(* Schneider Machine Expert - Basic project es3_4pompe_3max_6soglie_spegnimento_graduale_semplice, file version 3.0.0.0 *)
(* ProjectInformations: Name=New project *)

HARDWARE
  Cpu 0: TM221C40R
  EthernetConfiguration: NetworkName=M221, IpAllocationMode=FixedAddress, IpAddress=0.0.0.0, SubnetMask=0.0.0.0
  SerialLineConfiguration: Baud=Baud19200, Parity=ParityEven, DataBits=DataBits8, StopBits=StopBits1, PhysicalMedium=PhysicalMediumRs485, TransmissionMode=TransmissionModeModbusRtu, SlaveId=1, Addressing=SlaveAddressing
  MastTask: UsePeriodScanMode=false, PeriodScan=100
  FastTask: Period=255
  CpuBehavior: StartingMode=StartAsPreviousState, AutoSaveRamOnEeprom=true, WatchdogPeriod=250

SYMBOLS  (address, symbol, comment, settings)
  %M0       P1_USABILE
  %M1       P2_USABILE
  %M2       P1_COMANDATA  "Stesso valore di P1_CMD. Permette di identificare gli edges, visto che P1_CMD non può farlo."
  %M3       P2_COMANDATA  "Stesso valore di P2_CMD. Permette di identificare gli edges, visto che P2_CMD non può farlo."
  %M4       P3_USABILE
  %M5       P4_USABILE
  %M6       P3_COMANDATA
  %M7       P4_COMANDATA
  %M8       ESISTE_PROX_POMPA_CON_MINOR_ORE  "Nel loop, può non esistere una prossima pompa usabile e non comandata con il minor numero ore."
  %M9       ORA_E_00  "E' mezzanotte?"
  %M10      DECISO_ORDINE  "In intervallo in cui alternare le pompe per altern. giorn., è stata deciso quale sarà prossima pompa con minor ore?"
  %M11      PRIMA_POMPA_COMANDATA  "La prima pompa dell'ordine è stata effettivamente comandata quando serviva?"
  %M12      SECONDA_POMPA_COMANDATA  "La seconda pompa dell'ordine è stata effettivamente comandata quando serviva?"
  %M13      TERZA_POMPA_COMANDATA  "La terza pompa dell'ordine è stata effettivamente comandata quando serviva?"
  %S6       SB_TB1S  "Time base of 1 s generated by an internal clock"
  %MW0      NUM_POMPE_DA_COMANDARE  "Numero di pompe da comandare in base alle soglie raggiunte."
  %MW1      NUM_POMPE_COMANDATE  "Numero di pompe effettivamente comandate, in base alle loro disponibilità."
  %MW2      NUM_POMPE  "Numero di pompe totali."
  %MW3      ULTIMO_MINOR_SECONDI_LAVORATI  "Ultimi secondi lavorati più piccoli (valore temporaneo, da usare solo nel loop)."
  %MW4      PROSSIMA_POMPA_DA_COMANDARE  "Numero da 1 a NUM_POMPE che indica la prossima pompa da comandare."
  %MW5      POMPA_ATTUALE_LOOP  "Pompa attuale nel loop."
  %MW6      NUM_POMPE_COMANDATE_MAX  "Num"
  %MW7      CONTA_POMPE_COMANDATE_MAX  "Da usare in loop e da resettare.  Assume il valore da 1 fino a NUM_POMPE_COMANDATE_MAX."
  %MW8      ORDINE_PRIMA_POMPA
  %MW9      ORDINE_SECONDA_POMPA
  %MW10     ORDINE_TERZA_POMPA
  %C0       CONTATORE_P1_SECONDI_LAVORATI  [Preset=0]
  %C1       CONTATORE_P2_SECONDI_LAVORATI  [Preset=0]
  %C2       CONTATORE_P3_SECONDI_LAVORATI  [Preset=0]
  %C3       CONTATORE_P4_SECONDI_LAVORATI  [Preset=0]
  %I0.0     P1_AUTO
  %I0.1     P1_MOTO
  %I0.2     P1_ANOMALIA
  %I0.3     P2_AUTO
  %I0.4     P2_MOTO
  %I0.5     P2_ANOMALIA
  %I0.6     LVL_MIN1
  %I0.7     LVL_MAX1
  %I0.8     LVL_MAX2
  %I0.9     P3_AUTO
  %I0.10    P3_MOTO
  %I0.11    P3_ANOMALIA
  %I0.12    P4_AUTO
  %I0.13    P4_MOTO
  %I0.14    P4_ANOMALIA
  %I0.15    LVL_MAX3
  %I0.16    LVL_MIN2
  %I0.17    LVL_MIN3
  %Q0.0     P1_CMD
  %Q0.1     P2_CMD
  %Q0.2     P3_CMD
  %Q0.3     P4_CMD

POU Main
  (* SectionNumber=1 *)

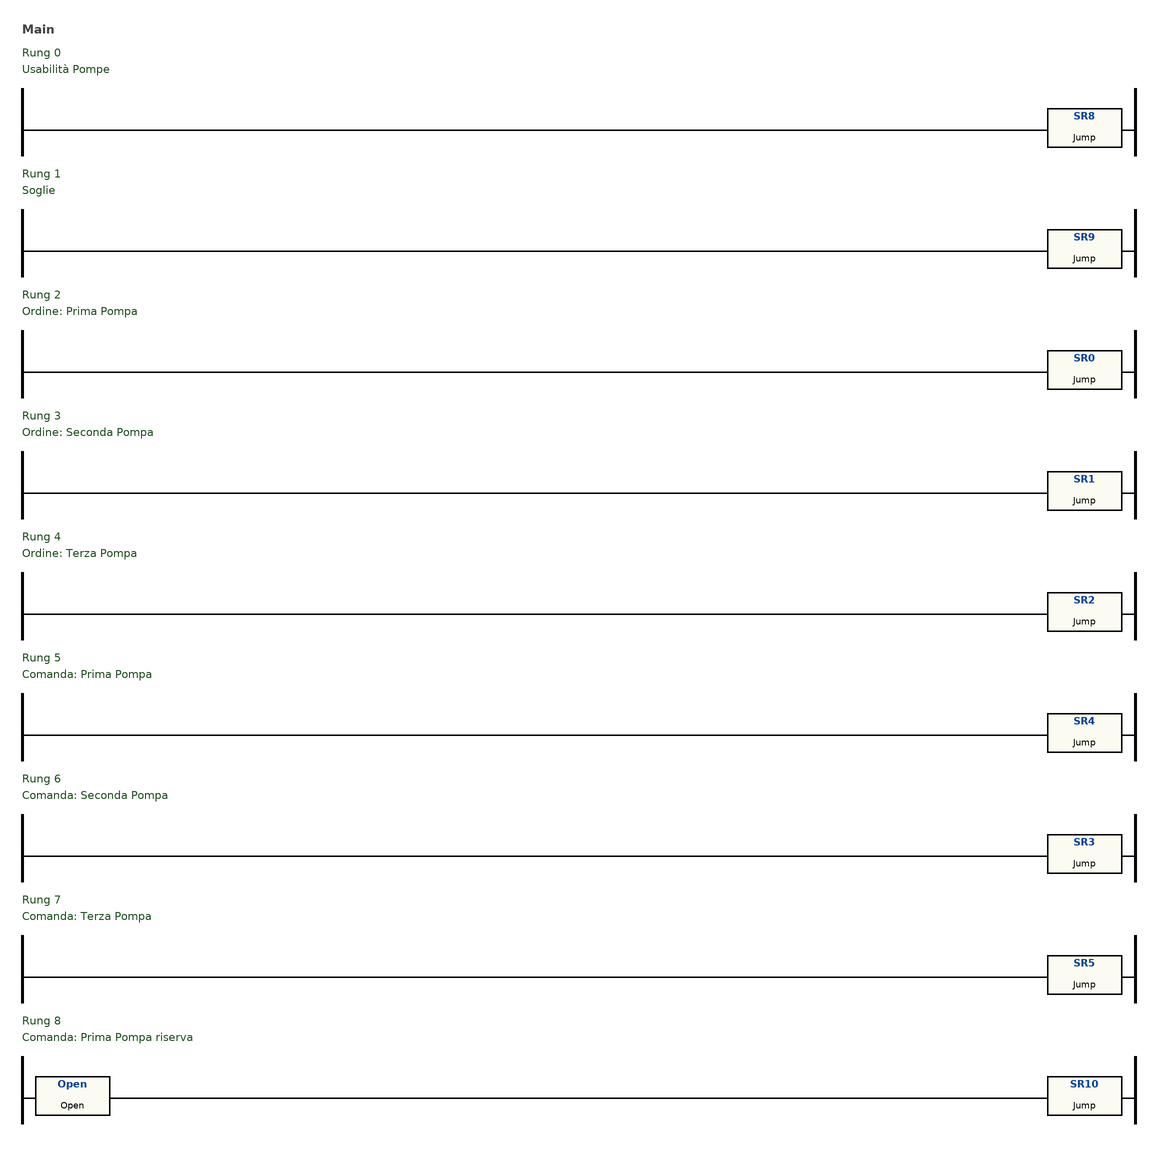

// Rung 0
// Usabilità Pompe
  LD 1
  SR8
  // as ST:
  //   SR8();

// Rung 1
// Soglie
  LD 1
  SR9
  // as ST:
  //   SR9();

// Rung 2
// Ordine: Prima Pompa
  LD 1
  SR0
  // as ST:
  //   SR0();

// Rung 3
// Ordine: Seconda Pompa
  LD 1
  SR1
  // as ST:
  //   SR1();

// Rung 4
// Ordine: Terza Pompa
  LD 1
  SR2
  // as ST:
  //   SR2();

// Rung 5
// Comanda: Prima Pompa
  LD 1
  SR4
  // as ST:
  //   SR4();

// Rung 6
// Comanda: Seconda Pompa
  LD 1
  SR3
  // as ST:
  //   SR3();

// Rung 7
// Comanda: Terza Pompa
  LD 1
  SR5
  // as ST:
  //   SR5();

// Rung 8
// Comanda: Prima Pompa riserva
  LD 0
  SR10
  // as ST:
  //   IF FALSE THEN SR10(); END_IF;

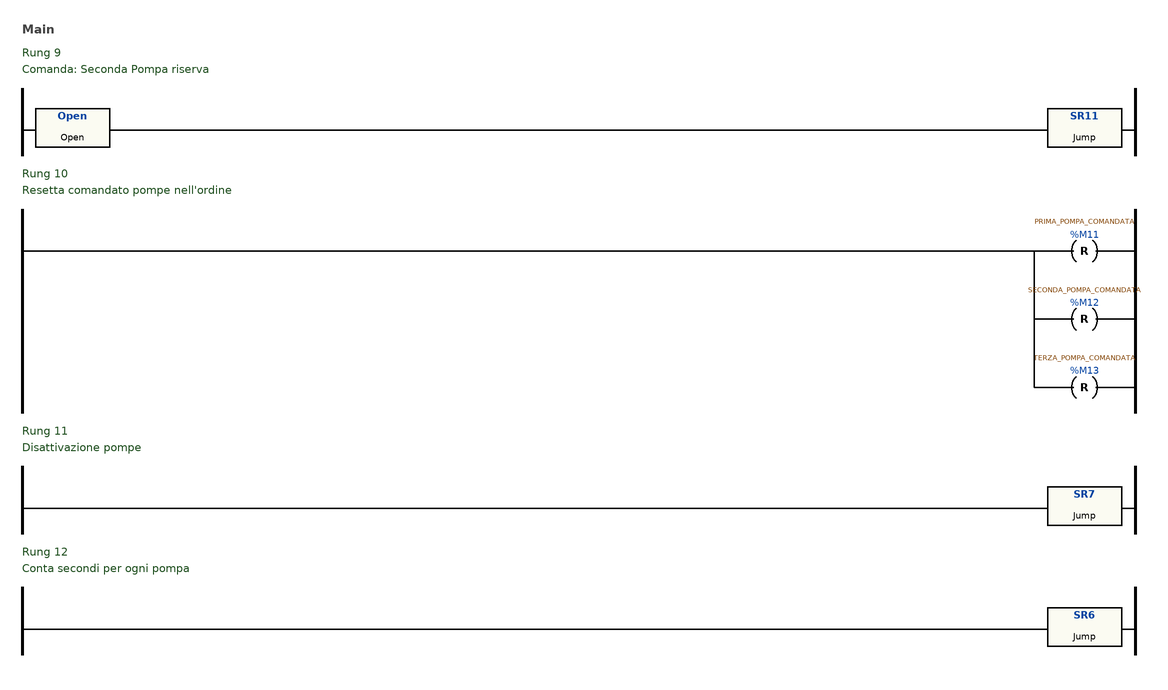

// Rung 9
// Comanda: Seconda Pompa riserva
  LD 0
  SR11
  // as ST:
  //   IF FALSE THEN SR11(); END_IF;

// Rung 10
// Resetta comandato pompe nell'ordine
  LD 1
  R %M11                  (* PRIMA_POMPA_COMANDATA *)
  R %M12                  (* SECONDA_POMPA_COMANDATA *)
  R %M13                  (* TERZA_POMPA_COMANDATA *)
  // as ST:
  //   PRIMA_POMPA_COMANDATA := FALSE;
  //   SECONDA_POMPA_COMANDATA := FALSE;
  //   TERZA_POMPA_COMANDATA := FALSE;

// Rung 11
// Disattivazione pompe
  LD 1
  SR7
  // as ST:
  //   SR7();

// Rung 12
// Conta secondi per ogni pompa
  LD 1
  SR6
  // as ST:
  //   SR6();

Subroutine Ordine: Prima Pompa
  (* SectionNumber=2, Number=0 *)

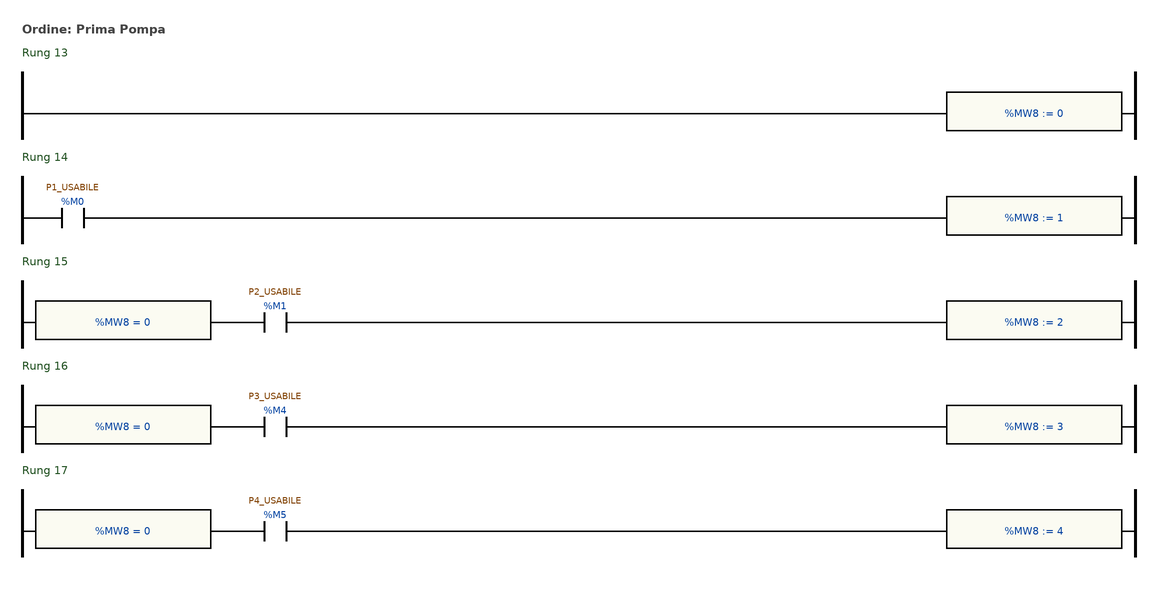

// Rung 13
  LD 1
  [ %MW8 := 0 ]           (* ORDINE_PRIMA_POMPA *)
  // as ST:
  //   ORDINE_PRIMA_POMPA := 0;

// Rung 14
  LD %M0                  (* P1_USABILE *)
  [ %MW8 := 1 ]           (* ORDINE_PRIMA_POMPA *)
  // as ST:
  //   IF P1_USABILE THEN ORDINE_PRIMA_POMPA := 1; END_IF;

// Rung 15
  LD [ %MW8 = 0 ]         (* ORDINE_PRIMA_POMPA *)
  AND %M1                 (* P2_USABILE *)
  [ %MW8 := 2 ]           (* ORDINE_PRIMA_POMPA *)
  // as ST:
  //   IF ORDINE_PRIMA_POMPA = 0 AND P2_USABILE THEN ORDINE_PRIMA_POMPA := 2; END_IF;

// Rung 16
  LD [ %MW8 = 0 ]         (* ORDINE_PRIMA_POMPA *)
  AND %M4                 (* P3_USABILE *)
  [ %MW8 := 3 ]           (* ORDINE_PRIMA_POMPA *)
  // as ST:
  //   IF ORDINE_PRIMA_POMPA = 0 AND P3_USABILE THEN ORDINE_PRIMA_POMPA := 3; END_IF;

// Rung 17
  LD [ %MW8 = 0 ]         (* ORDINE_PRIMA_POMPA *)
  AND %M5                 (* P4_USABILE *)
  [ %MW8 := 4 ]           (* ORDINE_PRIMA_POMPA *)
  // as ST:
  //   IF ORDINE_PRIMA_POMPA = 0 AND P4_USABILE THEN ORDINE_PRIMA_POMPA := 4; END_IF;

Subroutine Ordine: Seconda Pompa
  (* SectionNumber=3, Number=1 *)

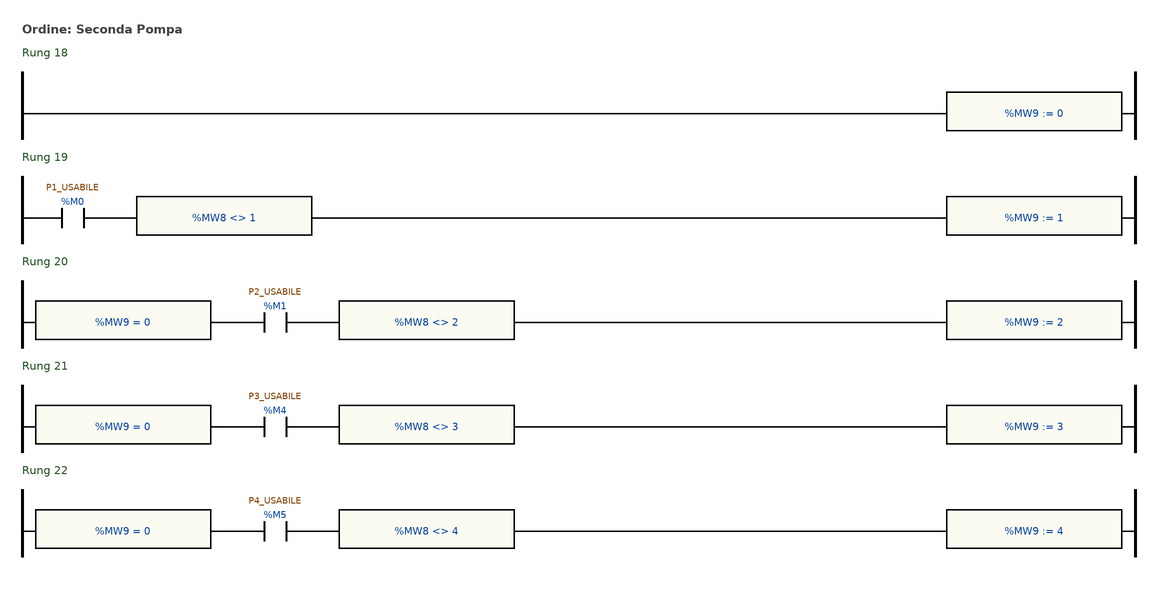

// Rung 18
  LD 1
  [ %MW9 := 0 ]           (* ORDINE_SECONDA_POMPA *)
  // as ST:
  //   ORDINE_SECONDA_POMPA := 0;

// Rung 19
  LD %M0                  (* P1_USABILE *)
  AND [ %MW8 <> 1 ]       (* ORDINE_PRIMA_POMPA *)
  [ %MW9 := 1 ]           (* ORDINE_SECONDA_POMPA *)
  // as ST:
  //   IF P1_USABILE AND ORDINE_PRIMA_POMPA <> 1 THEN ORDINE_SECONDA_POMPA := 1; END_IF;

// Rung 20
  LD [ %MW9 = 0 ]         (* ORDINE_SECONDA_POMPA *)
  AND %M1                 (* P2_USABILE *)
  AND [ %MW8 <> 2 ]       (* ORDINE_PRIMA_POMPA *)
  [ %MW9 := 2 ]           (* ORDINE_SECONDA_POMPA *)
  // as ST:
  //   IF ORDINE_SECONDA_POMPA = 0 AND P2_USABILE AND ORDINE_PRIMA_POMPA <> 2 THEN ORDINE_SECONDA_POMPA := 2; END_IF;

// Rung 21
  LD [ %MW9 = 0 ]         (* ORDINE_SECONDA_POMPA *)
  AND %M4                 (* P3_USABILE *)
  AND [ %MW8 <> 3 ]       (* ORDINE_PRIMA_POMPA *)
  [ %MW9 := 3 ]           (* ORDINE_SECONDA_POMPA *)
  // as ST:
  //   IF ORDINE_SECONDA_POMPA = 0 AND P3_USABILE AND ORDINE_PRIMA_POMPA <> 3 THEN ORDINE_SECONDA_POMPA := 3; END_IF;

// Rung 22
  LD [ %MW9 = 0 ]         (* ORDINE_SECONDA_POMPA *)
  AND %M5                 (* P4_USABILE *)
  AND [ %MW8 <> 4 ]       (* ORDINE_PRIMA_POMPA *)
  [ %MW9 := 4 ]           (* ORDINE_SECONDA_POMPA *)
  // as ST:
  //   IF ORDINE_SECONDA_POMPA = 0 AND P4_USABILE AND ORDINE_PRIMA_POMPA <> 4 THEN ORDINE_SECONDA_POMPA := 4; END_IF;

Subroutine Ordine: Terza Pompa
  (* SectionNumber=4, Number=2 *)

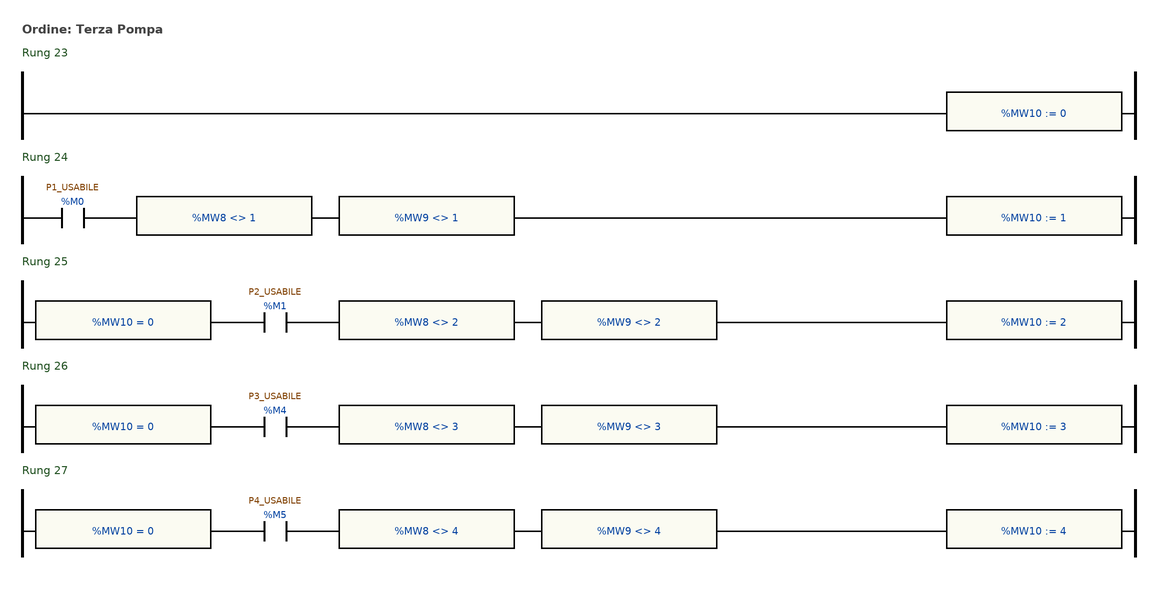

// Rung 23
  LD 1
  [ %MW10 := 0 ]          (* ORDINE_TERZA_POMPA *)
  // as ST:
  //   ORDINE_TERZA_POMPA := 0;

// Rung 24
  LD %M0                  (* P1_USABILE *)
  AND [ %MW8 <> 1 ]       (* ORDINE_PRIMA_POMPA *)
  AND [ %MW9 <> 1 ]       (* ORDINE_SECONDA_POMPA *)
  [ %MW10 := 1 ]          (* ORDINE_TERZA_POMPA *)
  // as ST:
  //   IF P1_USABILE AND ORDINE_PRIMA_POMPA <> 1 AND ORDINE_SECONDA_POMPA <> 1 THEN ORDINE_TERZA_POMPA := 1; END_IF;

// Rung 25
  LD [ %MW10 = 0 ]        (* ORDINE_TERZA_POMPA *)
  AND %M1                 (* P2_USABILE *)
  AND [ %MW8 <> 2 ]       (* ORDINE_PRIMA_POMPA *)
  AND [ %MW9 <> 2 ]       (* ORDINE_SECONDA_POMPA *)
  [ %MW10 := 2 ]          (* ORDINE_TERZA_POMPA *)
  // as ST:
  //   IF ORDINE_TERZA_POMPA = 0 AND P2_USABILE AND ORDINE_PRIMA_POMPA <> 2 AND ORDINE_SECONDA_POMPA <> 2 THEN ORDINE_TERZA_POMPA := 2; END_IF;

// Rung 26
  LD [ %MW10 = 0 ]        (* ORDINE_TERZA_POMPA *)
  AND %M4                 (* P3_USABILE *)
  AND [ %MW8 <> 3 ]       (* ORDINE_PRIMA_POMPA *)
  AND [ %MW9 <> 3 ]       (* ORDINE_SECONDA_POMPA *)
  [ %MW10 := 3 ]          (* ORDINE_TERZA_POMPA *)
  // as ST:
  //   IF ORDINE_TERZA_POMPA = 0 AND P3_USABILE AND ORDINE_PRIMA_POMPA <> 3 AND ORDINE_SECONDA_POMPA <> 3 THEN ORDINE_TERZA_POMPA := 3; END_IF;

// Rung 27
  LD [ %MW10 = 0 ]        (* ORDINE_TERZA_POMPA *)
  AND %M5                 (* P4_USABILE *)
  AND [ %MW8 <> 4 ]       (* ORDINE_PRIMA_POMPA *)
  AND [ %MW9 <> 4 ]       (* ORDINE_SECONDA_POMPA *)
  [ %MW10 := 4 ]          (* ORDINE_TERZA_POMPA *)
  // as ST:
  //   IF ORDINE_TERZA_POMPA = 0 AND P4_USABILE AND ORDINE_PRIMA_POMPA <> 4 AND ORDINE_SECONDA_POMPA <> 4 THEN ORDINE_TERZA_POMPA := 4; END_IF;

Subroutine Comanda: Prima Pompa
  (* SectionNumber=5, Number=4 *)

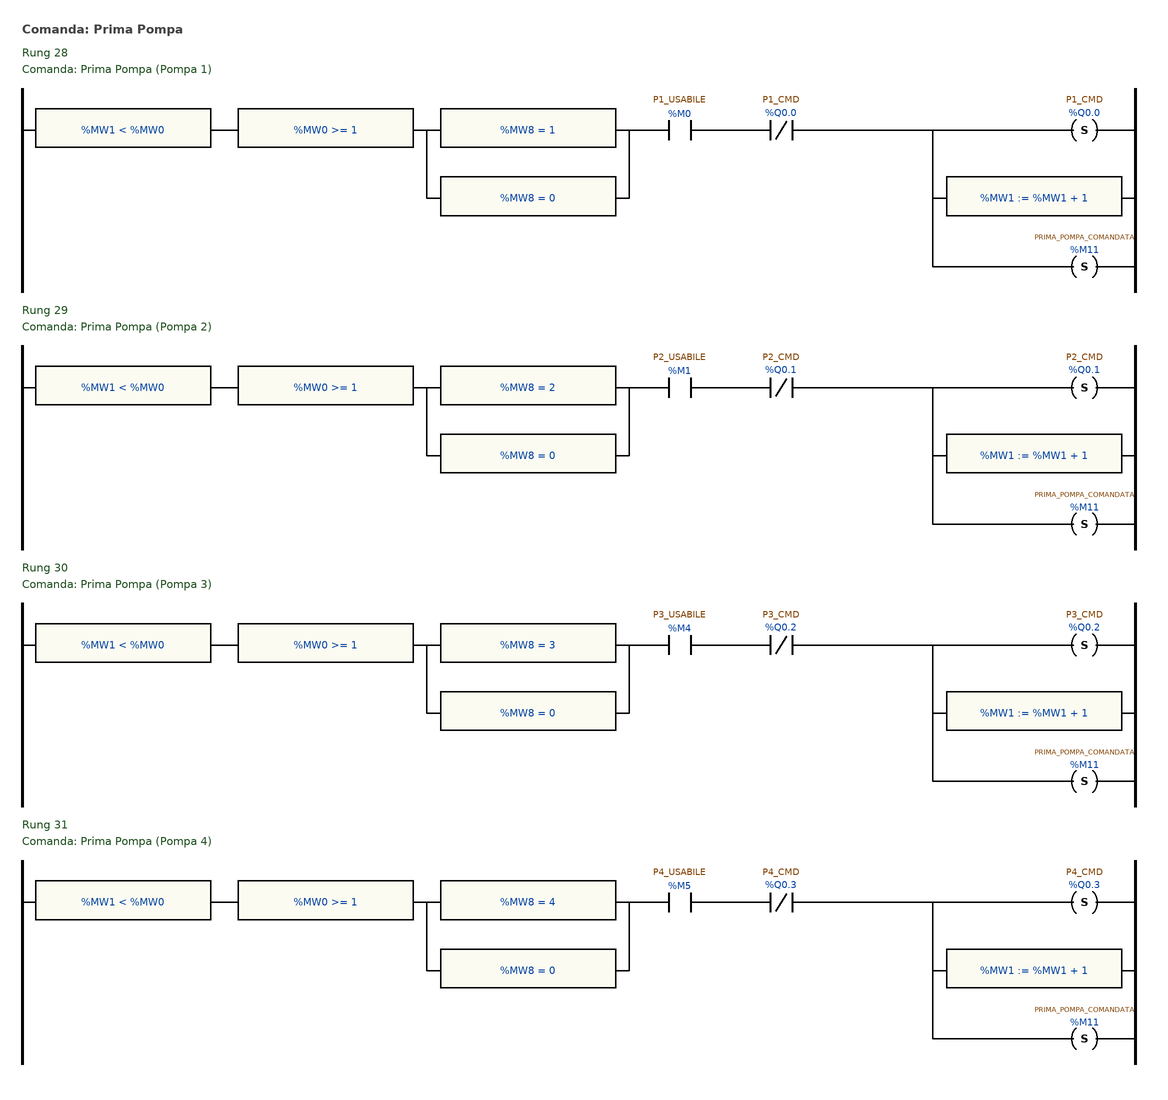

// Rung 28
// Comanda: Prima Pompa (Pompa 1)
  LD [ %MW1 < %MW0 ]      (* NUM_POMPE_COMANDATE, NUM_POMPE_DA_COMANDARE *)
  AND [ %MW0 >= 1 ]       (* NUM_POMPE_DA_COMANDARE *)
  AND( [ %MW8 = 1 ]       (* ORDINE_PRIMA_POMPA *)
  OR [ %MW8 = 0 ]         (* ORDINE_PRIMA_POMPA *)
  )
  AND %M0                 (* P1_USABILE *)
  ANDN %Q0.0              (* P1_CMD *)
  S %Q0.0                 (* P1_CMD *)
  [ %MW1 := %MW1 + 1 ]    (* NUM_POMPE_COMANDATE, NUM_POMPE_COMANDATE *)
  S %M11                  (* PRIMA_POMPA_COMANDATA *)
  // as ST:
  //   _t1 := NUM_POMPE_COMANDATE < NUM_POMPE_DA_COMANDARE AND NUM_POMPE_DA_COMANDARE >= 1 AND (ORDINE_PRIMA_POMPA = 1 OR ORDINE_PRIMA_POMPA = 0) AND P1_USABILE AND NOT P1_CMD;
  //   IF _t1 THEN P1_CMD := TRUE; END_IF;
  //   IF _t1 THEN NUM_POMPE_COMANDATE := NUM_POMPE_COMANDATE + 1; END_IF;
  //   IF _t1 THEN PRIMA_POMPA_COMANDATA := TRUE; END_IF;

// Rung 29
// Comanda: Prima Pompa (Pompa 2)
  LD [ %MW1 < %MW0 ]      (* NUM_POMPE_COMANDATE, NUM_POMPE_DA_COMANDARE *)
  AND [ %MW0 >= 1 ]       (* NUM_POMPE_DA_COMANDARE *)
  AND( [ %MW8 = 2 ]       (* ORDINE_PRIMA_POMPA *)
  OR [ %MW8 = 0 ]         (* ORDINE_PRIMA_POMPA *)
  )
  AND %M1                 (* P2_USABILE *)
  ANDN %Q0.1              (* P2_CMD *)
  S %Q0.1                 (* P2_CMD *)
  [ %MW1 := %MW1 + 1 ]    (* NUM_POMPE_COMANDATE, NUM_POMPE_COMANDATE *)
  S %M11                  (* PRIMA_POMPA_COMANDATA *)
  // as ST:
  //   _t1 := NUM_POMPE_COMANDATE < NUM_POMPE_DA_COMANDARE AND NUM_POMPE_DA_COMANDARE >= 1 AND (ORDINE_PRIMA_POMPA = 2 OR ORDINE_PRIMA_POMPA = 0) AND P2_USABILE AND NOT P2_CMD;
  //   IF _t1 THEN P2_CMD := TRUE; END_IF;
  //   IF _t1 THEN NUM_POMPE_COMANDATE := NUM_POMPE_COMANDATE + 1; END_IF;
  //   IF _t1 THEN PRIMA_POMPA_COMANDATA := TRUE; END_IF;

// Rung 30
// Comanda: Prima Pompa (Pompa 3)
  LD [ %MW1 < %MW0 ]      (* NUM_POMPE_COMANDATE, NUM_POMPE_DA_COMANDARE *)
  AND [ %MW0 >= 1 ]       (* NUM_POMPE_DA_COMANDARE *)
  AND( [ %MW8 = 3 ]       (* ORDINE_PRIMA_POMPA *)
  OR [ %MW8 = 0 ]         (* ORDINE_PRIMA_POMPA *)
  )
  AND %M4                 (* P3_USABILE *)
  ANDN %Q0.2              (* P3_CMD *)
  S %Q0.2                 (* P3_CMD *)
  [ %MW1 := %MW1 + 1 ]    (* NUM_POMPE_COMANDATE, NUM_POMPE_COMANDATE *)
  S %M11                  (* PRIMA_POMPA_COMANDATA *)
  // as ST:
  //   _t1 := NUM_POMPE_COMANDATE < NUM_POMPE_DA_COMANDARE AND NUM_POMPE_DA_COMANDARE >= 1 AND (ORDINE_PRIMA_POMPA = 3 OR ORDINE_PRIMA_POMPA = 0) AND P3_USABILE AND NOT P3_CMD;
  //   IF _t1 THEN P3_CMD := TRUE; END_IF;
  //   IF _t1 THEN NUM_POMPE_COMANDATE := NUM_POMPE_COMANDATE + 1; END_IF;
  //   IF _t1 THEN PRIMA_POMPA_COMANDATA := TRUE; END_IF;

// Rung 31
// Comanda: Prima Pompa (Pompa 4)
  LD [ %MW1 < %MW0 ]      (* NUM_POMPE_COMANDATE, NUM_POMPE_DA_COMANDARE *)
  AND [ %MW0 >= 1 ]       (* NUM_POMPE_DA_COMANDARE *)
  AND( [ %MW8 = 4 ]       (* ORDINE_PRIMA_POMPA *)
  OR [ %MW8 = 0 ]         (* ORDINE_PRIMA_POMPA *)
  )
  AND %M5                 (* P4_USABILE *)
  ANDN %Q0.3              (* P4_CMD *)
  S %Q0.3                 (* P4_CMD *)
  [ %MW1 := %MW1 + 1 ]    (* NUM_POMPE_COMANDATE, NUM_POMPE_COMANDATE *)
  S %M11                  (* PRIMA_POMPA_COMANDATA *)
  // as ST:
  //   _t1 := NUM_POMPE_COMANDATE < NUM_POMPE_DA_COMANDARE AND NUM_POMPE_DA_COMANDARE >= 1 AND (ORDINE_PRIMA_POMPA = 4 OR ORDINE_PRIMA_POMPA = 0) AND P4_USABILE AND NOT P4_CMD;
  //   IF _t1 THEN P4_CMD := TRUE; END_IF;
  //   IF _t1 THEN NUM_POMPE_COMANDATE := NUM_POMPE_COMANDATE + 1; END_IF;
  //   IF _t1 THEN PRIMA_POMPA_COMANDATA := TRUE; END_IF;

Subroutine Comanda: Seconda Pompa
  (* SectionNumber=6, Number=3 *)

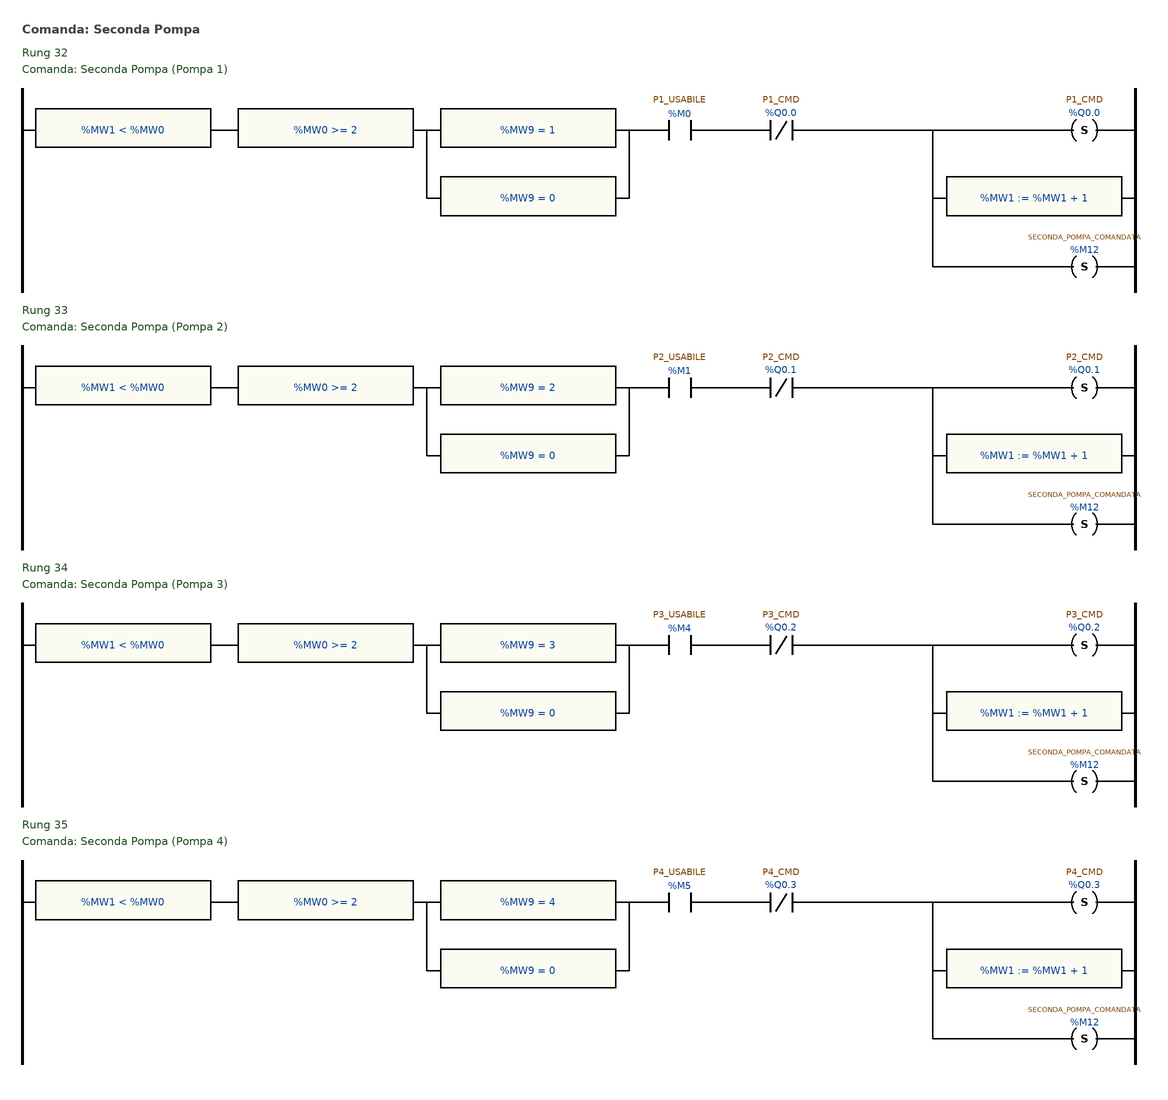

// Rung 32
// Comanda: Seconda Pompa (Pompa 1)
  LD [ %MW1 < %MW0 ]      (* NUM_POMPE_COMANDATE, NUM_POMPE_DA_COMANDARE *)
  AND [ %MW0 >= 2 ]       (* NUM_POMPE_DA_COMANDARE *)
  AND( [ %MW9 = 1 ]       (* ORDINE_SECONDA_POMPA *)
  OR [ %MW9 = 0 ]         (* ORDINE_SECONDA_POMPA *)
  )
  AND %M0                 (* P1_USABILE *)
  ANDN %Q0.0              (* P1_CMD *)
  S %Q0.0                 (* P1_CMD *)
  [ %MW1 := %MW1 + 1 ]    (* NUM_POMPE_COMANDATE, NUM_POMPE_COMANDATE *)
  S %M12                  (* SECONDA_POMPA_COMANDATA *)
  // as ST:
  //   _t1 := NUM_POMPE_COMANDATE < NUM_POMPE_DA_COMANDARE AND NUM_POMPE_DA_COMANDARE >= 2 AND (ORDINE_SECONDA_POMPA = 1 OR ORDINE_SECONDA_POMPA = 0) AND P1_USABILE AND NOT P1_CMD;
  //   IF _t1 THEN P1_CMD := TRUE; END_IF;
  //   IF _t1 THEN NUM_POMPE_COMANDATE := NUM_POMPE_COMANDATE + 1; END_IF;
  //   IF _t1 THEN SECONDA_POMPA_COMANDATA := TRUE; END_IF;

// Rung 33
// Comanda: Seconda Pompa (Pompa 2)
  LD [ %MW1 < %MW0 ]      (* NUM_POMPE_COMANDATE, NUM_POMPE_DA_COMANDARE *)
  AND [ %MW0 >= 2 ]       (* NUM_POMPE_DA_COMANDARE *)
  AND( [ %MW9 = 2 ]       (* ORDINE_SECONDA_POMPA *)
  OR [ %MW9 = 0 ]         (* ORDINE_SECONDA_POMPA *)
  )
  AND %M1                 (* P2_USABILE *)
  ANDN %Q0.1              (* P2_CMD *)
  S %Q0.1                 (* P2_CMD *)
  [ %MW1 := %MW1 + 1 ]    (* NUM_POMPE_COMANDATE, NUM_POMPE_COMANDATE *)
  S %M12                  (* SECONDA_POMPA_COMANDATA *)
  // as ST:
  //   _t1 := NUM_POMPE_COMANDATE < NUM_POMPE_DA_COMANDARE AND NUM_POMPE_DA_COMANDARE >= 2 AND (ORDINE_SECONDA_POMPA = 2 OR ORDINE_SECONDA_POMPA = 0) AND P2_USABILE AND NOT P2_CMD;
  //   IF _t1 THEN P2_CMD := TRUE; END_IF;
  //   IF _t1 THEN NUM_POMPE_COMANDATE := NUM_POMPE_COMANDATE + 1; END_IF;
  //   IF _t1 THEN SECONDA_POMPA_COMANDATA := TRUE; END_IF;

// Rung 34
// Comanda: Seconda Pompa (Pompa 3)
  LD [ %MW1 < %MW0 ]      (* NUM_POMPE_COMANDATE, NUM_POMPE_DA_COMANDARE *)
  AND [ %MW0 >= 2 ]       (* NUM_POMPE_DA_COMANDARE *)
  AND( [ %MW9 = 3 ]       (* ORDINE_SECONDA_POMPA *)
  OR [ %MW9 = 0 ]         (* ORDINE_SECONDA_POMPA *)
  )
  AND %M4                 (* P3_USABILE *)
  ANDN %Q0.2              (* P3_CMD *)
  S %Q0.2                 (* P3_CMD *)
  [ %MW1 := %MW1 + 1 ]    (* NUM_POMPE_COMANDATE, NUM_POMPE_COMANDATE *)
  S %M12                  (* SECONDA_POMPA_COMANDATA *)
  // as ST:
  //   _t1 := NUM_POMPE_COMANDATE < NUM_POMPE_DA_COMANDARE AND NUM_POMPE_DA_COMANDARE >= 2 AND (ORDINE_SECONDA_POMPA = 3 OR ORDINE_SECONDA_POMPA = 0) AND P3_USABILE AND NOT P3_CMD;
  //   IF _t1 THEN P3_CMD := TRUE; END_IF;
  //   IF _t1 THEN NUM_POMPE_COMANDATE := NUM_POMPE_COMANDATE + 1; END_IF;
  //   IF _t1 THEN SECONDA_POMPA_COMANDATA := TRUE; END_IF;

// Rung 35
// Comanda: Seconda Pompa (Pompa 4)
  LD [ %MW1 < %MW0 ]      (* NUM_POMPE_COMANDATE, NUM_POMPE_DA_COMANDARE *)
  AND [ %MW0 >= 2 ]       (* NUM_POMPE_DA_COMANDARE *)
  AND( [ %MW9 = 4 ]       (* ORDINE_SECONDA_POMPA *)
  OR [ %MW9 = 0 ]         (* ORDINE_SECONDA_POMPA *)
  )
  AND %M5                 (* P4_USABILE *)
  ANDN %Q0.3              (* P4_CMD *)
  S %Q0.3                 (* P4_CMD *)
  [ %MW1 := %MW1 + 1 ]    (* NUM_POMPE_COMANDATE, NUM_POMPE_COMANDATE *)
  S %M12                  (* SECONDA_POMPA_COMANDATA *)
  // as ST:
  //   _t1 := NUM_POMPE_COMANDATE < NUM_POMPE_DA_COMANDARE AND NUM_POMPE_DA_COMANDARE >= 2 AND (ORDINE_SECONDA_POMPA = 4 OR ORDINE_SECONDA_POMPA = 0) AND P4_USABILE AND NOT P4_CMD;
  //   IF _t1 THEN P4_CMD := TRUE; END_IF;
  //   IF _t1 THEN NUM_POMPE_COMANDATE := NUM_POMPE_COMANDATE + 1; END_IF;
  //   IF _t1 THEN SECONDA_POMPA_COMANDATA := TRUE; END_IF;

Subroutine Comanda: Terza Pompa
  (* SectionNumber=7, Number=5 *)

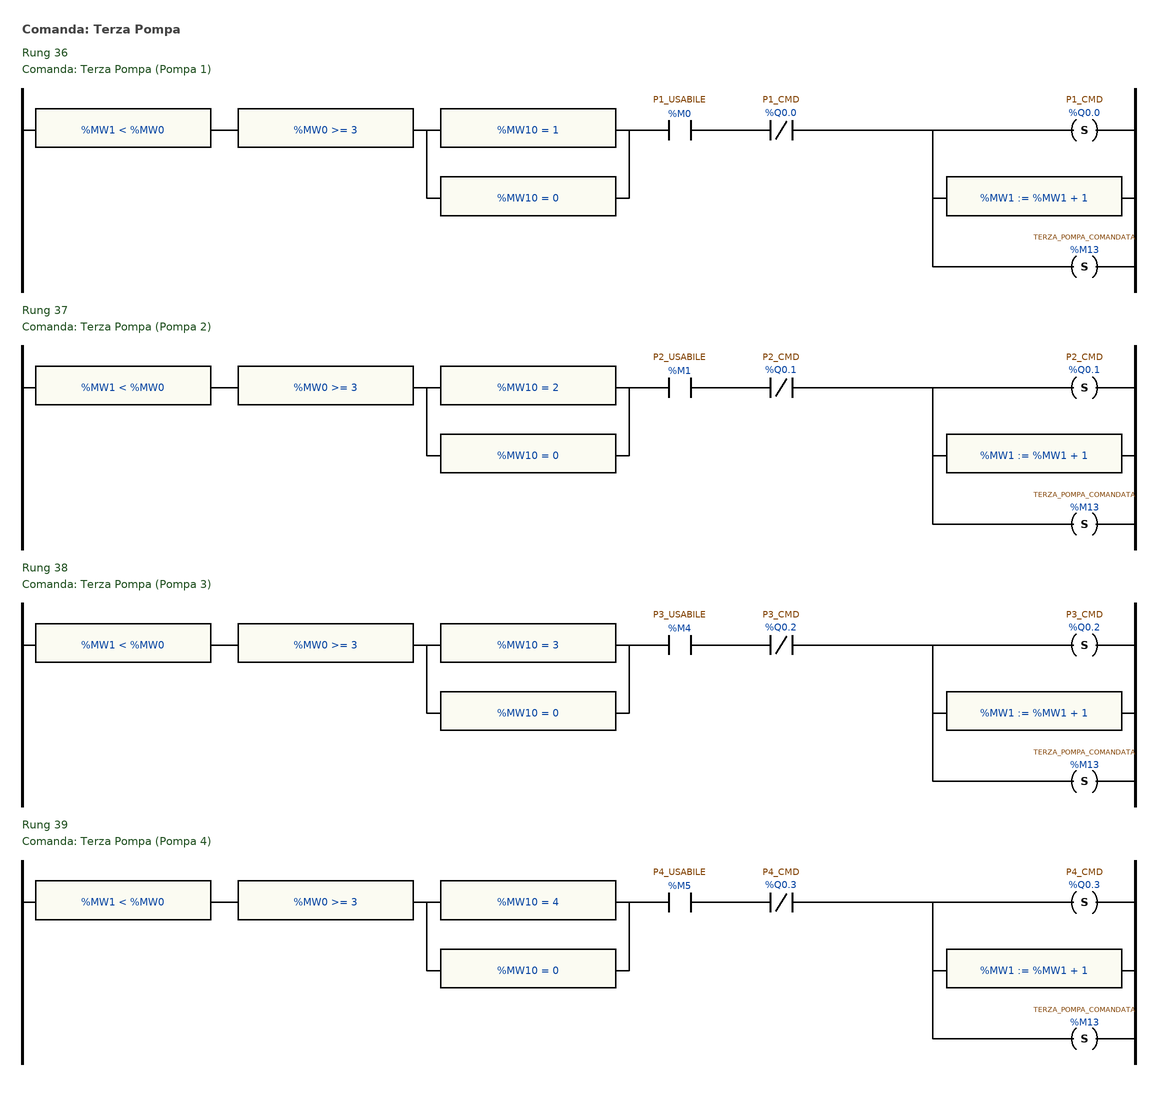

// Rung 36
// Comanda: Terza Pompa (Pompa 1)
  LD [ %MW1 < %MW0 ]      (* NUM_POMPE_COMANDATE, NUM_POMPE_DA_COMANDARE *)
  AND [ %MW0 >= 3 ]       (* NUM_POMPE_DA_COMANDARE *)
  AND( [ %MW10 = 1 ]      (* ORDINE_TERZA_POMPA *)
  OR [ %MW10 = 0 ]        (* ORDINE_TERZA_POMPA *)
  )
  AND %M0                 (* P1_USABILE *)
  ANDN %Q0.0              (* P1_CMD *)
  S %Q0.0                 (* P1_CMD *)
  [ %MW1 := %MW1 + 1 ]    (* NUM_POMPE_COMANDATE, NUM_POMPE_COMANDATE *)
  S %M13                  (* TERZA_POMPA_COMANDATA *)
  // as ST:
  //   _t1 := NUM_POMPE_COMANDATE < NUM_POMPE_DA_COMANDARE AND NUM_POMPE_DA_COMANDARE >= 3 AND (ORDINE_TERZA_POMPA = 1 OR ORDINE_TERZA_POMPA = 0) AND P1_USABILE AND NOT P1_CMD;
  //   IF _t1 THEN P1_CMD := TRUE; END_IF;
  //   IF _t1 THEN NUM_POMPE_COMANDATE := NUM_POMPE_COMANDATE + 1; END_IF;
  //   IF _t1 THEN TERZA_POMPA_COMANDATA := TRUE; END_IF;

// Rung 37
// Comanda: Terza Pompa (Pompa 2)
  LD [ %MW1 < %MW0 ]      (* NUM_POMPE_COMANDATE, NUM_POMPE_DA_COMANDARE *)
  AND [ %MW0 >= 3 ]       (* NUM_POMPE_DA_COMANDARE *)
  AND( [ %MW10 = 2 ]      (* ORDINE_TERZA_POMPA *)
  OR [ %MW10 = 0 ]        (* ORDINE_TERZA_POMPA *)
  )
  AND %M1                 (* P2_USABILE *)
  ANDN %Q0.1              (* P2_CMD *)
  S %Q0.1                 (* P2_CMD *)
  [ %MW1 := %MW1 + 1 ]    (* NUM_POMPE_COMANDATE, NUM_POMPE_COMANDATE *)
  S %M13                  (* TERZA_POMPA_COMANDATA *)
  // as ST:
  //   _t1 := NUM_POMPE_COMANDATE < NUM_POMPE_DA_COMANDARE AND NUM_POMPE_DA_COMANDARE >= 3 AND (ORDINE_TERZA_POMPA = 2 OR ORDINE_TERZA_POMPA = 0) AND P2_USABILE AND NOT P2_CMD;
  //   IF _t1 THEN P2_CMD := TRUE; END_IF;
  //   IF _t1 THEN NUM_POMPE_COMANDATE := NUM_POMPE_COMANDATE + 1; END_IF;
  //   IF _t1 THEN TERZA_POMPA_COMANDATA := TRUE; END_IF;

// Rung 38
// Comanda: Terza Pompa (Pompa 3)
  LD [ %MW1 < %MW0 ]      (* NUM_POMPE_COMANDATE, NUM_POMPE_DA_COMANDARE *)
  AND [ %MW0 >= 3 ]       (* NUM_POMPE_DA_COMANDARE *)
  AND( [ %MW10 = 3 ]      (* ORDINE_TERZA_POMPA *)
  OR [ %MW10 = 0 ]        (* ORDINE_TERZA_POMPA *)
  )
  AND %M4                 (* P3_USABILE *)
  ANDN %Q0.2              (* P3_CMD *)
  S %Q0.2                 (* P3_CMD *)
  [ %MW1 := %MW1 + 1 ]    (* NUM_POMPE_COMANDATE, NUM_POMPE_COMANDATE *)
  S %M13                  (* TERZA_POMPA_COMANDATA *)
  // as ST:
  //   _t1 := NUM_POMPE_COMANDATE < NUM_POMPE_DA_COMANDARE AND NUM_POMPE_DA_COMANDARE >= 3 AND (ORDINE_TERZA_POMPA = 3 OR ORDINE_TERZA_POMPA = 0) AND P3_USABILE AND NOT P3_CMD;
  //   IF _t1 THEN P3_CMD := TRUE; END_IF;
  //   IF _t1 THEN NUM_POMPE_COMANDATE := NUM_POMPE_COMANDATE + 1; END_IF;
  //   IF _t1 THEN TERZA_POMPA_COMANDATA := TRUE; END_IF;

// Rung 39
// Comanda: Terza Pompa (Pompa 4)
  LD [ %MW1 < %MW0 ]      (* NUM_POMPE_COMANDATE, NUM_POMPE_DA_COMANDARE *)
  AND [ %MW0 >= 3 ]       (* NUM_POMPE_DA_COMANDARE *)
  AND( [ %MW10 = 4 ]      (* ORDINE_TERZA_POMPA *)
  OR [ %MW10 = 0 ]        (* ORDINE_TERZA_POMPA *)
  )
  AND %M5                 (* P4_USABILE *)
  ANDN %Q0.3              (* P4_CMD *)
  S %Q0.3                 (* P4_CMD *)
  [ %MW1 := %MW1 + 1 ]    (* NUM_POMPE_COMANDATE, NUM_POMPE_COMANDATE *)
  S %M13                  (* TERZA_POMPA_COMANDATA *)
  // as ST:
  //   _t1 := NUM_POMPE_COMANDATE < NUM_POMPE_DA_COMANDARE AND NUM_POMPE_DA_COMANDARE >= 3 AND (ORDINE_TERZA_POMPA = 4 OR ORDINE_TERZA_POMPA = 0) AND P4_USABILE AND NOT P4_CMD;
  //   IF _t1 THEN P4_CMD := TRUE; END_IF;
  //   IF _t1 THEN NUM_POMPE_COMANDATE := NUM_POMPE_COMANDATE + 1; END_IF;
  //   IF _t1 THEN TERZA_POMPA_COMANDATA := TRUE; END_IF;

Subroutine Conta Secondi per Pompa
  (* SectionNumber=8, Number=6 *)

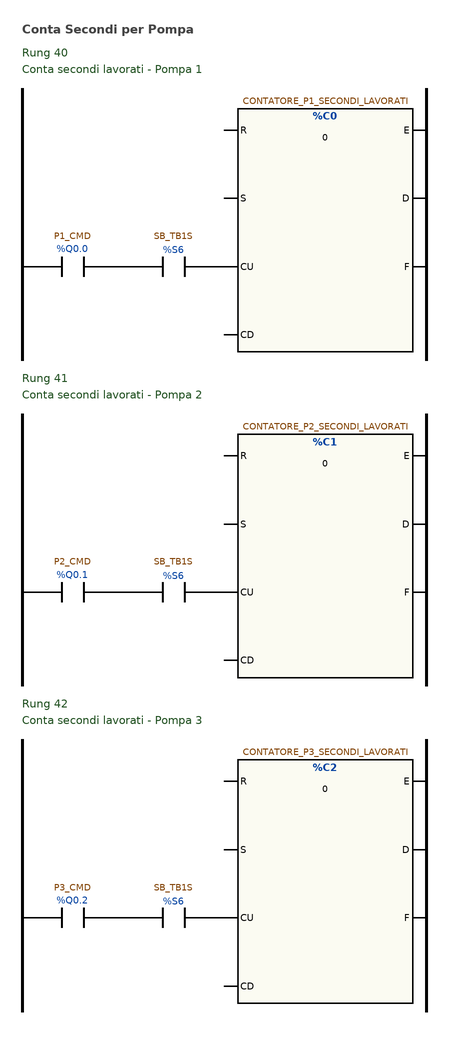

// Rung 40
// Conta secondi lavorati - Pompa 1
  BLK %C0                 (* CONTATORE_P1_SECONDI_LAVORATI *)
  LD %Q0.0                (* P1_CMD *)
  AND %S6                 (* SB_TB1S *)
  CU
  END_BLK
  // as ST:
  //   CONTATORE_P1_SECONDI_LAVORATI(CU := P1_CMD AND SB_TB1S);

// Rung 41
// Conta secondi lavorati - Pompa 2
  BLK %C1                 (* CONTATORE_P2_SECONDI_LAVORATI *)
  LD %Q0.1                (* P2_CMD *)
  AND %S6                 (* SB_TB1S *)
  CU
  END_BLK
  // as ST:
  //   CONTATORE_P2_SECONDI_LAVORATI(CU := P2_CMD AND SB_TB1S);

// Rung 42
// Conta secondi lavorati - Pompa 3
  BLK %C2                 (* CONTATORE_P3_SECONDI_LAVORATI *)
  LD %Q0.2                (* P3_CMD *)
  AND %S6                 (* SB_TB1S *)
  CU
  END_BLK
  // as ST:
  //   CONTATORE_P3_SECONDI_LAVORATI(CU := P3_CMD AND SB_TB1S);

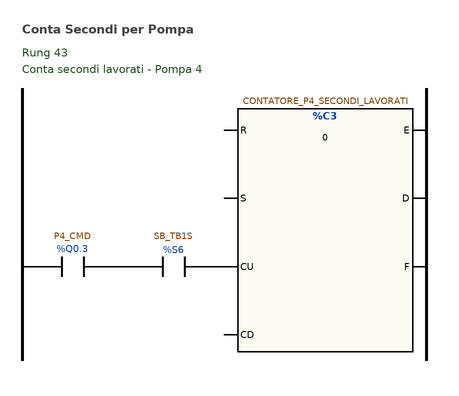

// Rung 43
// Conta secondi lavorati - Pompa 4
  BLK %C3                 (* CONTATORE_P4_SECONDI_LAVORATI *)
  LD %Q0.3                (* P4_CMD *)
  AND %S6                 (* SB_TB1S *)
  CU
  END_BLK
  // as ST:
  //   CONTATORE_P4_SECONDI_LAVORATI(CU := P4_CMD AND SB_TB1S);

Subroutine Disattivazione Pompe
  (* SectionNumber=9, Number=7 *)

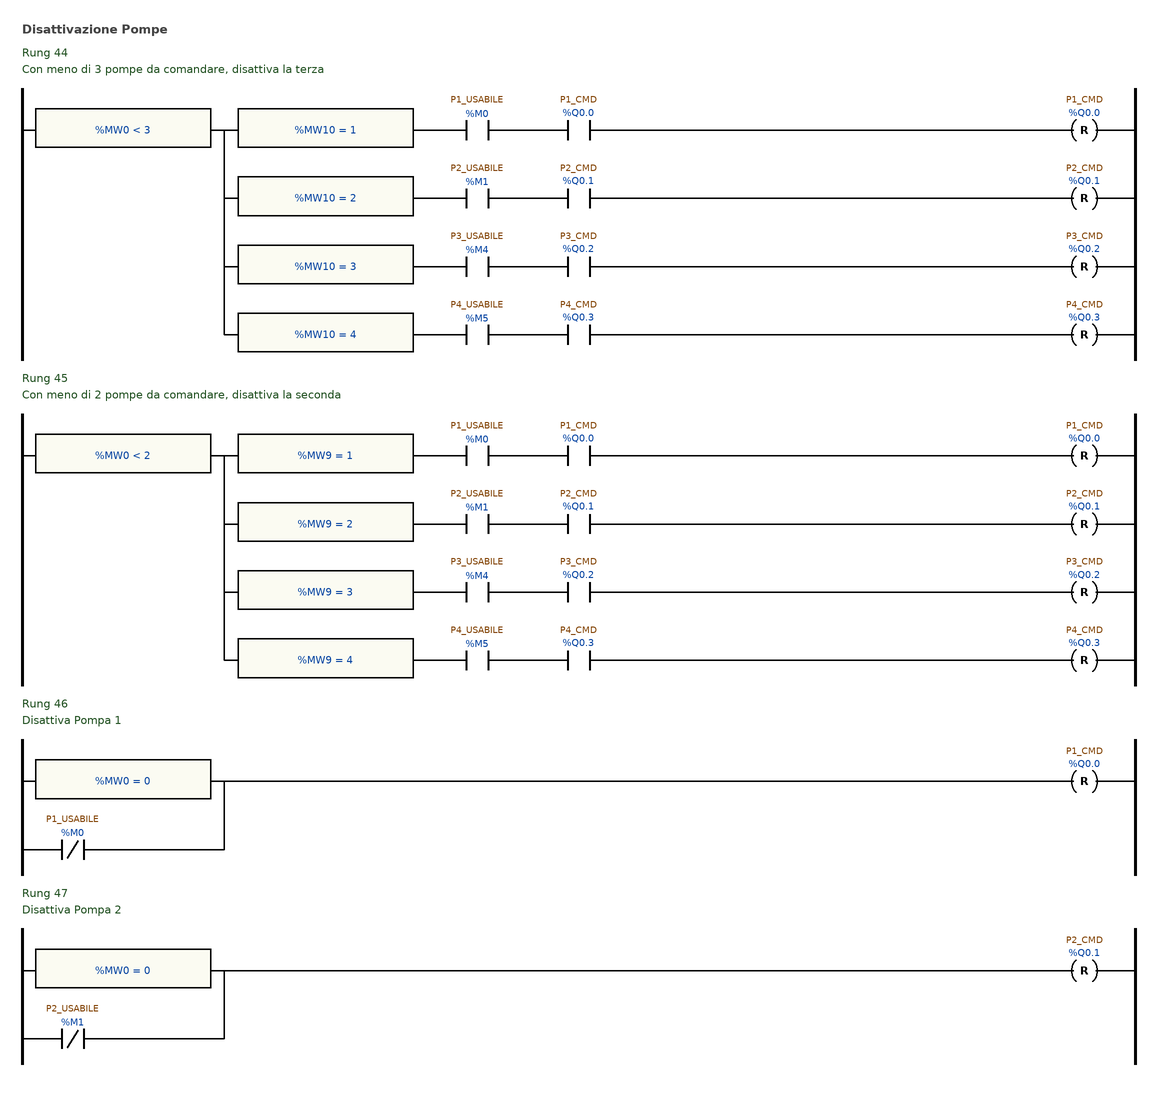

// Rung 44
// Con meno di 3 pompe da comandare, disattiva la terza
  LD [ %MW0 < 3 ]         (* NUM_POMPE_DA_COMANDARE *)
  MPS
  AND [ %MW10 = 1 ]       (* ORDINE_TERZA_POMPA *)
  AND %M0                 (* P1_USABILE *)
  AND %Q0.0               (* P1_CMD *)
  R %Q0.0                 (* P1_CMD *)
  MRD
  AND [ %MW10 = 2 ]       (* ORDINE_TERZA_POMPA *)
  AND %M1                 (* P2_USABILE *)
  AND %Q0.1               (* P2_CMD *)
  R %Q0.1                 (* P2_CMD *)
  MRD
  AND [ %MW10 = 3 ]       (* ORDINE_TERZA_POMPA *)
  AND %M4                 (* P3_USABILE *)
  AND %Q0.2               (* P3_CMD *)
  R %Q0.2                 (* P3_CMD *)
  MPP
  AND [ %MW10 = 4 ]       (* ORDINE_TERZA_POMPA *)
  AND %M5                 (* P4_USABILE *)
  AND %Q0.3               (* P4_CMD *)
  R %Q0.3                 (* P4_CMD *)
  // as ST:
  //   IF NUM_POMPE_DA_COMANDARE < 3 AND ORDINE_TERZA_POMPA = 1 AND P1_USABILE AND P1_CMD THEN P1_CMD := FALSE; END_IF;
  //   IF NUM_POMPE_DA_COMANDARE < 3 AND ORDINE_TERZA_POMPA = 2 AND P2_USABILE AND P2_CMD THEN P2_CMD := FALSE; END_IF;
  //   IF NUM_POMPE_DA_COMANDARE < 3 AND ORDINE_TERZA_POMPA = 3 AND P3_USABILE AND P3_CMD THEN P3_CMD := FALSE; END_IF;
  //   IF NUM_POMPE_DA_COMANDARE < 3 AND ORDINE_TERZA_POMPA = 4 AND P4_USABILE AND P4_CMD THEN P4_CMD := FALSE; END_IF;

// Rung 45
// Con meno di 2 pompe da comandare, disattiva la seconda
  LD [ %MW0 < 2 ]         (* NUM_POMPE_DA_COMANDARE *)
  MPS
  AND [ %MW9 = 1 ]        (* ORDINE_SECONDA_POMPA *)
  AND %M0                 (* P1_USABILE *)
  AND %Q0.0               (* P1_CMD *)
  R %Q0.0                 (* P1_CMD *)
  MRD
  AND [ %MW9 = 2 ]        (* ORDINE_SECONDA_POMPA *)
  AND %M1                 (* P2_USABILE *)
  AND %Q0.1               (* P2_CMD *)
  R %Q0.1                 (* P2_CMD *)
  MRD
  AND [ %MW9 = 3 ]        (* ORDINE_SECONDA_POMPA *)
  AND %M4                 (* P3_USABILE *)
  AND %Q0.2               (* P3_CMD *)
  R %Q0.2                 (* P3_CMD *)
  MPP
  AND [ %MW9 = 4 ]        (* ORDINE_SECONDA_POMPA *)
  AND %M5                 (* P4_USABILE *)
  AND %Q0.3               (* P4_CMD *)
  R %Q0.3                 (* P4_CMD *)
  // as ST:
  //   IF NUM_POMPE_DA_COMANDARE < 2 AND ORDINE_SECONDA_POMPA = 1 AND P1_USABILE AND P1_CMD THEN P1_CMD := FALSE; END_IF;
  //   IF NUM_POMPE_DA_COMANDARE < 2 AND ORDINE_SECONDA_POMPA = 2 AND P2_USABILE AND P2_CMD THEN P2_CMD := FALSE; END_IF;
  //   IF NUM_POMPE_DA_COMANDARE < 2 AND ORDINE_SECONDA_POMPA = 3 AND P3_USABILE AND P3_CMD THEN P3_CMD := FALSE; END_IF;
  //   IF NUM_POMPE_DA_COMANDARE < 2 AND ORDINE_SECONDA_POMPA = 4 AND P4_USABILE AND P4_CMD THEN P4_CMD := FALSE; END_IF;

// Rung 46
// Disattiva Pompa 1
  LD [ %MW0 = 0 ]         (* NUM_POMPE_DA_COMANDARE *)
  ORN %M0                 (* P1_USABILE *)
  R %Q0.0                 (* P1_CMD *)
  // as ST:
  //   IF NUM_POMPE_DA_COMANDARE = 0 OR NOT P1_USABILE THEN P1_CMD := FALSE; END_IF;

// Rung 47
// Disattiva Pompa 2
  LD [ %MW0 = 0 ]         (* NUM_POMPE_DA_COMANDARE *)
  ORN %M1                 (* P2_USABILE *)
  R %Q0.1                 (* P2_CMD *)
  // as ST:
  //   IF NUM_POMPE_DA_COMANDARE = 0 OR NOT P2_USABILE THEN P2_CMD := FALSE; END_IF;

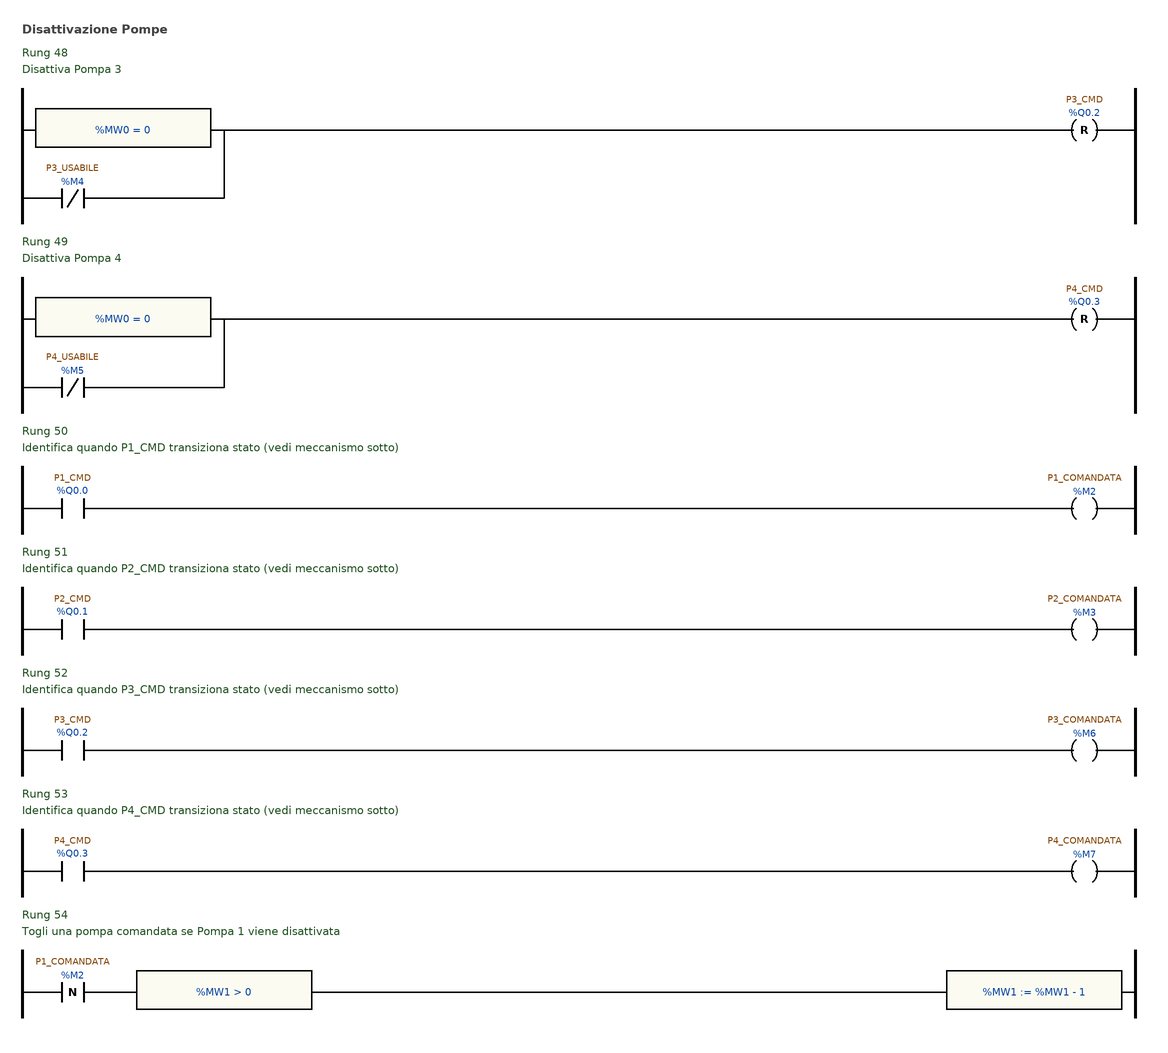

// Rung 48
// Disattiva Pompa 3
  LD [ %MW0 = 0 ]         (* NUM_POMPE_DA_COMANDARE *)
  ORN %M4                 (* P3_USABILE *)
  R %Q0.2                 (* P3_CMD *)
  // as ST:
  //   IF NUM_POMPE_DA_COMANDARE = 0 OR NOT P3_USABILE THEN P3_CMD := FALSE; END_IF;

// Rung 49
// Disattiva Pompa 4
  LD [ %MW0 = 0 ]         (* NUM_POMPE_DA_COMANDARE *)
  ORN %M5                 (* P4_USABILE *)
  R %Q0.3                 (* P4_CMD *)
  // as ST:
  //   IF NUM_POMPE_DA_COMANDARE = 0 OR NOT P4_USABILE THEN P4_CMD := FALSE; END_IF;

// Rung 50
// Identifica quando P1_CMD transiziona stato (vedi meccanismo sotto)
  LD %Q0.0                (* P1_CMD *)
  ST %M2                  (* P1_COMANDATA *)
  // as ST:
  //   P1_COMANDATA := P1_CMD;

// Rung 51
// Identifica quando P2_CMD transiziona stato (vedi meccanismo sotto)
  LD %Q0.1                (* P2_CMD *)
  ST %M3                  (* P2_COMANDATA *)
  // as ST:
  //   P2_COMANDATA := P2_CMD;

// Rung 52
// Identifica quando P3_CMD transiziona stato (vedi meccanismo sotto)
  LD %Q0.2                (* P3_CMD *)
  ST %M6                  (* P3_COMANDATA *)
  // as ST:
  //   P3_COMANDATA := P3_CMD;

// Rung 53
// Identifica quando P4_CMD transiziona stato (vedi meccanismo sotto)
  LD %Q0.3                (* P4_CMD *)
  ST %M7                  (* P4_COMANDATA *)
  // as ST:
  //   P4_COMANDATA := P4_CMD;

// Rung 54
// Togli una pompa comandata se Pompa 1 viene disattivata
  LDF %M2                 (* P1_COMANDATA *)
  AND [ %MW1 > 0 ]        (* NUM_POMPE_COMANDATE *)
  [ %MW1 := %MW1 - 1 ]    (* NUM_POMPE_COMANDATE, NUM_POMPE_COMANDATE *)
  // as ST:
  //   IF FALLING(P1_COMANDATA) AND NUM_POMPE_COMANDATE > 0 THEN NUM_POMPE_COMANDATE := NUM_POMPE_COMANDATE - 1; END_IF;

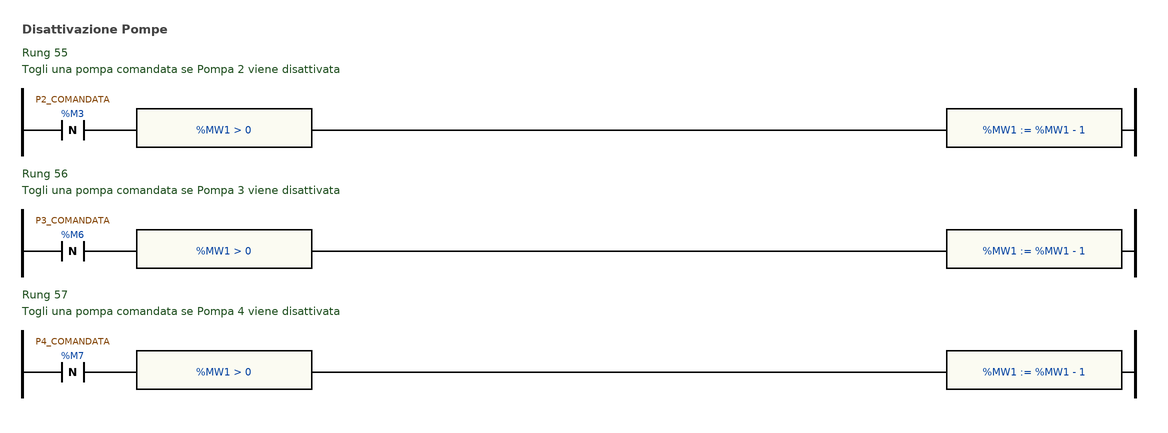

// Rung 55
// Togli una pompa comandata se Pompa 2 viene disattivata
  LDF %M3                 (* P2_COMANDATA *)
  AND [ %MW1 > 0 ]        (* NUM_POMPE_COMANDATE *)
  [ %MW1 := %MW1 - 1 ]    (* NUM_POMPE_COMANDATE, NUM_POMPE_COMANDATE *)
  // as ST:
  //   IF FALLING(P2_COMANDATA) AND NUM_POMPE_COMANDATE > 0 THEN NUM_POMPE_COMANDATE := NUM_POMPE_COMANDATE - 1; END_IF;

// Rung 56
// Togli una pompa comandata se Pompa 3 viene disattivata
  LDF %M6                 (* P3_COMANDATA *)
  AND [ %MW1 > 0 ]        (* NUM_POMPE_COMANDATE *)
  [ %MW1 := %MW1 - 1 ]    (* NUM_POMPE_COMANDATE, NUM_POMPE_COMANDATE *)
  // as ST:
  //   IF FALLING(P3_COMANDATA) AND NUM_POMPE_COMANDATE > 0 THEN NUM_POMPE_COMANDATE := NUM_POMPE_COMANDATE - 1; END_IF;

// Rung 57
// Togli una pompa comandata se Pompa 4 viene disattivata
  LDF %M7                 (* P4_COMANDATA *)
  AND [ %MW1 > 0 ]        (* NUM_POMPE_COMANDATE *)
  [ %MW1 := %MW1 - 1 ]    (* NUM_POMPE_COMANDATE, NUM_POMPE_COMANDATE *)
  // as ST:
  //   IF FALLING(P4_COMANDATA) AND NUM_POMPE_COMANDATE > 0 THEN NUM_POMPE_COMANDATE := NUM_POMPE_COMANDATE - 1; END_IF;

Subroutine Usabilità Pompe
  (* SectionNumber=10, Number=8 *)

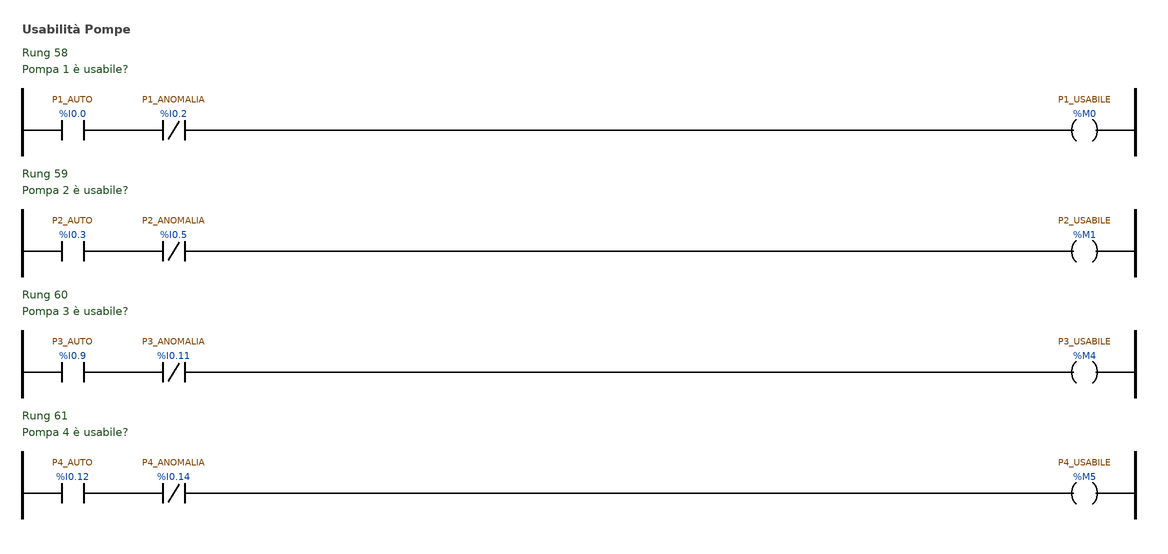

// Rung 58
// Pompa 1 è usabile?
  LD %I0.0                (* P1_AUTO *)
  ANDN %I0.2              (* P1_ANOMALIA *)
  ST %M0                  (* P1_USABILE *)
  // as ST:
  //   P1_USABILE := P1_AUTO AND NOT P1_ANOMALIA;

// Rung 59
// Pompa 2 è usabile?
  LD %I0.3                (* P2_AUTO *)
  ANDN %I0.5              (* P2_ANOMALIA *)
  ST %M1                  (* P2_USABILE *)
  // as ST:
  //   P2_USABILE := P2_AUTO AND NOT P2_ANOMALIA;

// Rung 60
// Pompa 3 è usabile?
  LD %I0.9                (* P3_AUTO *)
  ANDN %I0.11             (* P3_ANOMALIA *)
  ST %M4                  (* P3_USABILE *)
  // as ST:
  //   P3_USABILE := P3_AUTO AND NOT P3_ANOMALIA;

// Rung 61
// Pompa 4 è usabile?
  LD %I0.12               (* P4_AUTO *)
  ANDN %I0.14             (* P4_ANOMALIA *)
  ST %M5                  (* P4_USABILE *)
  // as ST:
  //   P4_USABILE := P4_AUTO AND NOT P4_ANOMALIA;

Subroutine Soglie
  (* SectionNumber=11, Number=9 *)

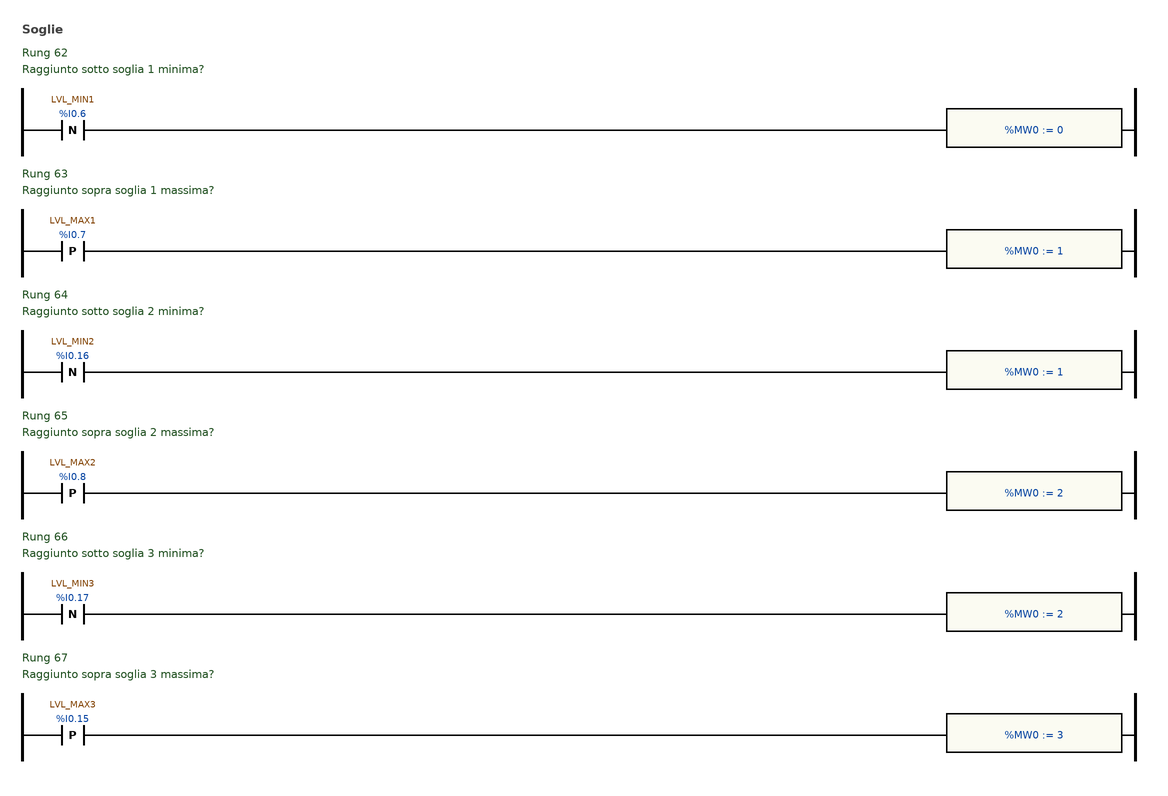

// Rung 62
// Raggiunto sotto soglia 1 minima?
  LDF %I0.6               (* LVL_MIN1 *)
  [ %MW0 := 0 ]           (* NUM_POMPE_DA_COMANDARE *)
  // as ST:
  //   IF FALLING(LVL_MIN1) THEN NUM_POMPE_DA_COMANDARE := 0; END_IF;

// Rung 63
// Raggiunto sopra soglia 1 massima?
  LDR %I0.7               (* LVL_MAX1 *)
  [ %MW0 := 1 ]           (* NUM_POMPE_DA_COMANDARE *)
  // as ST:
  //   IF RISING(LVL_MAX1) THEN NUM_POMPE_DA_COMANDARE := 1; END_IF;

// Rung 64
// Raggiunto sotto soglia 2 minima?
  LDF %I0.16              (* LVL_MIN2 *)
  [ %MW0 := 1 ]           (* NUM_POMPE_DA_COMANDARE *)
  // as ST:
  //   IF FALLING(LVL_MIN2) THEN NUM_POMPE_DA_COMANDARE := 1; END_IF;

// Rung 65
// Raggiunto sopra soglia 2 massima?
  LDR %I0.8               (* LVL_MAX2 *)
  [ %MW0 := 2 ]           (* NUM_POMPE_DA_COMANDARE *)
  // as ST:
  //   IF RISING(LVL_MAX2) THEN NUM_POMPE_DA_COMANDARE := 2; END_IF;

// Rung 66
// Raggiunto sotto soglia 3 minima?
  LDF %I0.17              (* LVL_MIN3 *)
  [ %MW0 := 2 ]           (* NUM_POMPE_DA_COMANDARE *)
  // as ST:
  //   IF FALLING(LVL_MIN3) THEN NUM_POMPE_DA_COMANDARE := 2; END_IF;

// Rung 67
// Raggiunto sopra soglia 3 massima?
  LDR %I0.15              (* LVL_MAX3 *)
  [ %MW0 := 3 ]           (* NUM_POMPE_DA_COMANDARE *)
  // as ST:
  //   IF RISING(LVL_MAX3) THEN NUM_POMPE_DA_COMANDARE := 3; END_IF;

Subroutine Comanda: Prima Pompa riserva
  (* SectionNumber=12, Number=10 *)

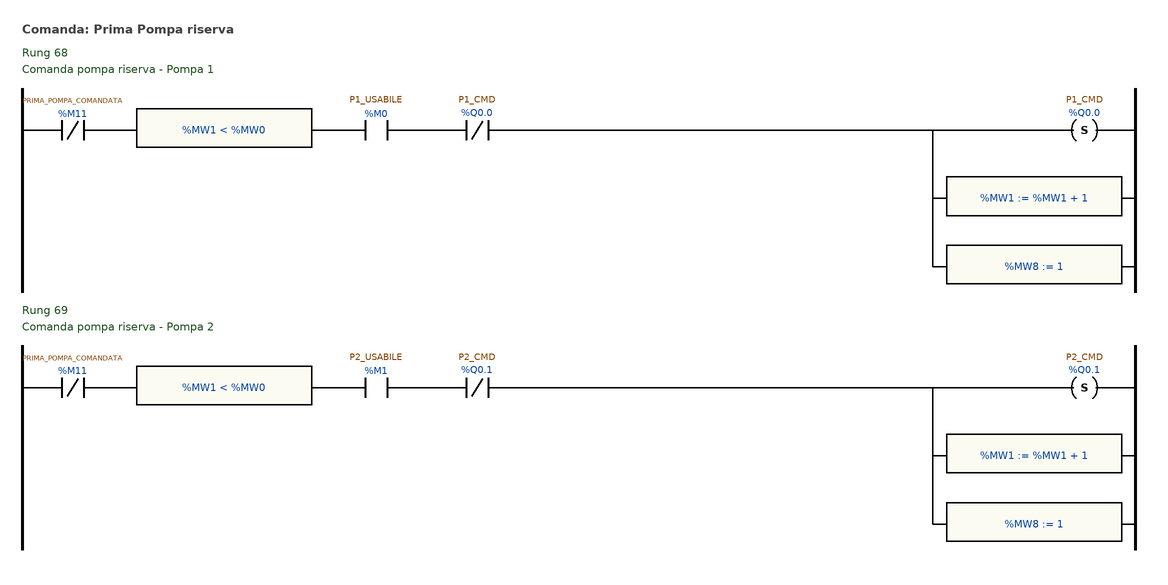

// Rung 68
// Comanda pompa riserva - Pompa 1
  LDN %M11                (* PRIMA_POMPA_COMANDATA *)
  AND [ %MW1 < %MW0 ]     (* NUM_POMPE_COMANDATE, NUM_POMPE_DA_COMANDARE *)
  AND %M0                 (* P1_USABILE *)
  ANDN %Q0.0              (* P1_CMD *)
  S %Q0.0                 (* P1_CMD *)
  [ %MW1 := %MW1 + 1 ]    (* NUM_POMPE_COMANDATE, NUM_POMPE_COMANDATE *)
  [ %MW8 := 1 ]           (* ORDINE_PRIMA_POMPA *)
  // as ST:
  //   _t1 := NOT PRIMA_POMPA_COMANDATA AND NUM_POMPE_COMANDATE < NUM_POMPE_DA_COMANDARE AND P1_USABILE AND NOT P1_CMD;
  //   IF _t1 THEN P1_CMD := TRUE; END_IF;
  //   IF _t1 THEN NUM_POMPE_COMANDATE := NUM_POMPE_COMANDATE + 1; END_IF;
  //   IF _t1 THEN ORDINE_PRIMA_POMPA := 1; END_IF;

// Rung 69
// Comanda pompa riserva - Pompa 2
  LDN %M11                (* PRIMA_POMPA_COMANDATA *)
  AND [ %MW1 < %MW0 ]     (* NUM_POMPE_COMANDATE, NUM_POMPE_DA_COMANDARE *)
  AND %M1                 (* P2_USABILE *)
  ANDN %Q0.1              (* P2_CMD *)
  S %Q0.1                 (* P2_CMD *)
  [ %MW1 := %MW1 + 1 ]    (* NUM_POMPE_COMANDATE, NUM_POMPE_COMANDATE *)
  [ %MW8 := 1 ]           (* ORDINE_PRIMA_POMPA *)
  // as ST:
  //   _t1 := NOT PRIMA_POMPA_COMANDATA AND NUM_POMPE_COMANDATE < NUM_POMPE_DA_COMANDARE AND P2_USABILE AND NOT P2_CMD;
  //   IF _t1 THEN P2_CMD := TRUE; END_IF;
  //   IF _t1 THEN NUM_POMPE_COMANDATE := NUM_POMPE_COMANDATE + 1; END_IF;
  //   IF _t1 THEN ORDINE_PRIMA_POMPA := 1; END_IF;

Subroutine Comanda: Seconda Pompa riserva
  (* SectionNumber=13, Number=11 *)

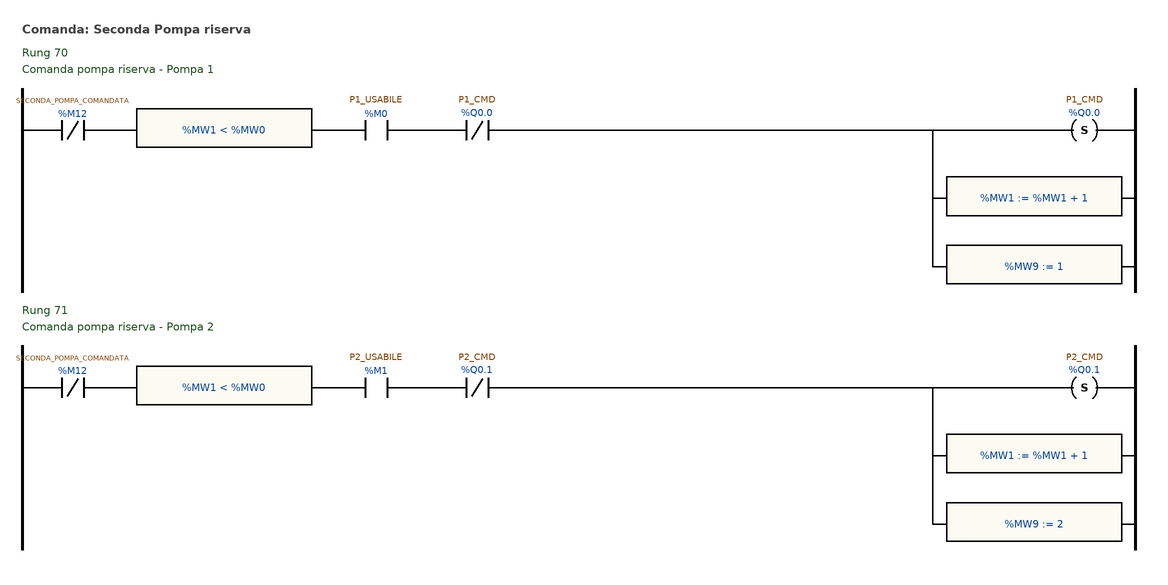

// Rung 70
// Comanda pompa riserva - Pompa 1
  LDN %M12                (* SECONDA_POMPA_COMANDATA *)
  AND [ %MW1 < %MW0 ]     (* NUM_POMPE_COMANDATE, NUM_POMPE_DA_COMANDARE *)
  AND %M0                 (* P1_USABILE *)
  ANDN %Q0.0              (* P1_CMD *)
  S %Q0.0                 (* P1_CMD *)
  [ %MW1 := %MW1 + 1 ]    (* NUM_POMPE_COMANDATE, NUM_POMPE_COMANDATE *)
  [ %MW9 := 1 ]           (* ORDINE_SECONDA_POMPA *)
  // as ST:
  //   _t1 := NOT SECONDA_POMPA_COMANDATA AND NUM_POMPE_COMANDATE < NUM_POMPE_DA_COMANDARE AND P1_USABILE AND NOT P1_CMD;
  //   IF _t1 THEN P1_CMD := TRUE; END_IF;
  //   IF _t1 THEN NUM_POMPE_COMANDATE := NUM_POMPE_COMANDATE + 1; END_IF;
  //   IF _t1 THEN ORDINE_SECONDA_POMPA := 1; END_IF;

// Rung 71
// Comanda pompa riserva - Pompa 2
  LDN %M12                (* SECONDA_POMPA_COMANDATA *)
  AND [ %MW1 < %MW0 ]     (* NUM_POMPE_COMANDATE, NUM_POMPE_DA_COMANDARE *)
  AND %M1                 (* P2_USABILE *)
  ANDN %Q0.1              (* P2_CMD *)
  S %Q0.1                 (* P2_CMD *)
  [ %MW1 := %MW1 + 1 ]    (* NUM_POMPE_COMANDATE, NUM_POMPE_COMANDATE *)
  [ %MW9 := 2 ]           (* ORDINE_SECONDA_POMPA *)
  // as ST:
  //   _t1 := NOT SECONDA_POMPA_COMANDATA AND NUM_POMPE_COMANDATE < NUM_POMPE_DA_COMANDARE AND P2_USABILE AND NOT P2_CMD;
  //   IF _t1 THEN P2_CMD := TRUE; END_IF;
  //   IF _t1 THEN NUM_POMPE_COMANDATE := NUM_POMPE_COMANDATE + 1; END_IF;
  //   IF _t1 THEN ORDINE_SECONDA_POMPA := 2; END_IF;

Subroutine Comanda: Terza Pompa riserva
  (* SectionNumber=14, Number=12 *)

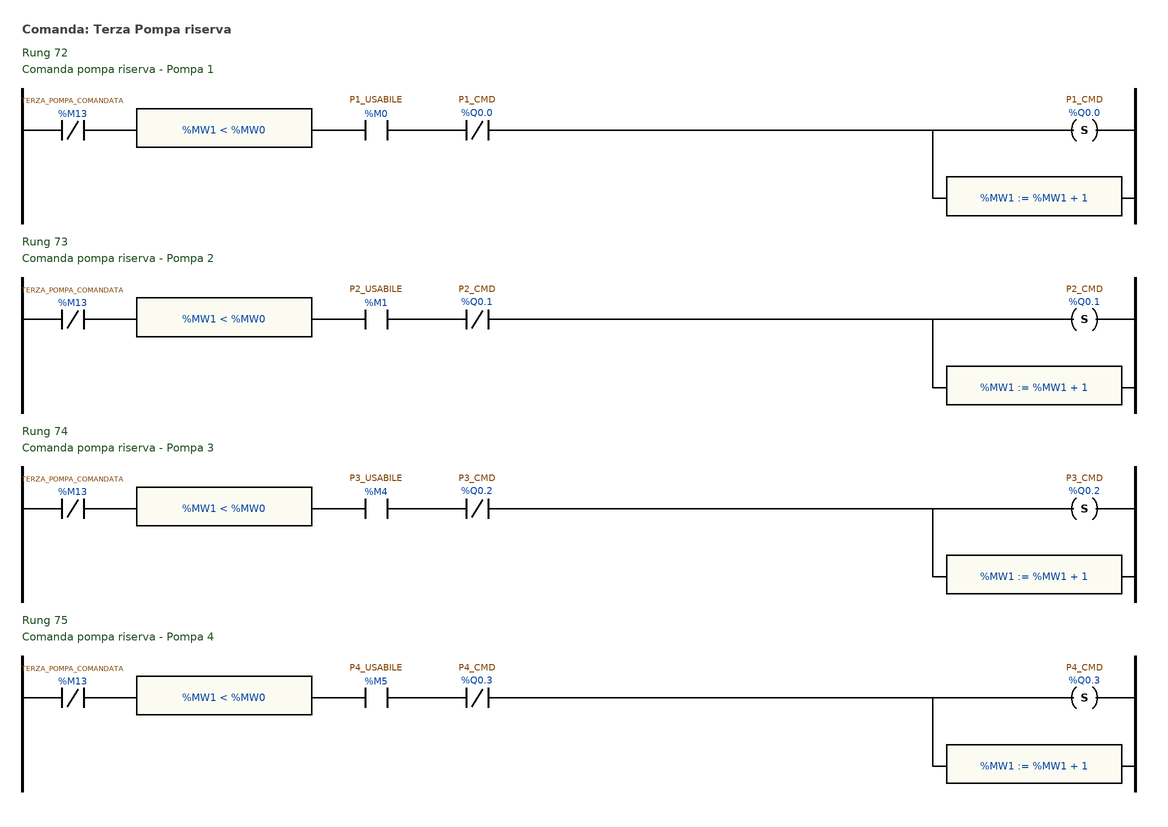

// Rung 72
// Comanda pompa riserva - Pompa 1
  LDN %M13                (* TERZA_POMPA_COMANDATA *)
  AND [ %MW1 < %MW0 ]     (* NUM_POMPE_COMANDATE, NUM_POMPE_DA_COMANDARE *)
  AND %M0                 (* P1_USABILE *)
  ANDN %Q0.0              (* P1_CMD *)
  S %Q0.0                 (* P1_CMD *)
  [ %MW1 := %MW1 + 1 ]    (* NUM_POMPE_COMANDATE, NUM_POMPE_COMANDATE *)
  // as ST:
  //   _t1 := NOT TERZA_POMPA_COMANDATA AND NUM_POMPE_COMANDATE < NUM_POMPE_DA_COMANDARE AND P1_USABILE AND NOT P1_CMD;
  //   IF _t1 THEN P1_CMD := TRUE; END_IF;
  //   IF _t1 THEN NUM_POMPE_COMANDATE := NUM_POMPE_COMANDATE + 1; END_IF;

// Rung 73
// Comanda pompa riserva - Pompa 2
  LDN %M13                (* TERZA_POMPA_COMANDATA *)
  AND [ %MW1 < %MW0 ]     (* NUM_POMPE_COMANDATE, NUM_POMPE_DA_COMANDARE *)
  AND %M1                 (* P2_USABILE *)
  ANDN %Q0.1              (* P2_CMD *)
  S %Q0.1                 (* P2_CMD *)
  [ %MW1 := %MW1 + 1 ]    (* NUM_POMPE_COMANDATE, NUM_POMPE_COMANDATE *)
  // as ST:
  //   _t1 := NOT TERZA_POMPA_COMANDATA AND NUM_POMPE_COMANDATE < NUM_POMPE_DA_COMANDARE AND P2_USABILE AND NOT P2_CMD;
  //   IF _t1 THEN P2_CMD := TRUE; END_IF;
  //   IF _t1 THEN NUM_POMPE_COMANDATE := NUM_POMPE_COMANDATE + 1; END_IF;

// Rung 74
// Comanda pompa riserva - Pompa 3
  LDN %M13                (* TERZA_POMPA_COMANDATA *)
  AND [ %MW1 < %MW0 ]     (* NUM_POMPE_COMANDATE, NUM_POMPE_DA_COMANDARE *)
  AND %M4                 (* P3_USABILE *)
  ANDN %Q0.2              (* P3_CMD *)
  S %Q0.2                 (* P3_CMD *)
  [ %MW1 := %MW1 + 1 ]    (* NUM_POMPE_COMANDATE, NUM_POMPE_COMANDATE *)
  // as ST:
  //   _t1 := NOT TERZA_POMPA_COMANDATA AND NUM_POMPE_COMANDATE < NUM_POMPE_DA_COMANDARE AND P3_USABILE AND NOT P3_CMD;
  //   IF _t1 THEN P3_CMD := TRUE; END_IF;
  //   IF _t1 THEN NUM_POMPE_COMANDATE := NUM_POMPE_COMANDATE + 1; END_IF;

// Rung 75
// Comanda pompa riserva - Pompa 4
  LDN %M13                (* TERZA_POMPA_COMANDATA *)
  AND [ %MW1 < %MW0 ]     (* NUM_POMPE_COMANDATE, NUM_POMPE_DA_COMANDARE *)
  AND %M5                 (* P4_USABILE *)
  ANDN %Q0.3              (* P4_CMD *)
  S %Q0.3                 (* P4_CMD *)
  [ %MW1 := %MW1 + 1 ]    (* NUM_POMPE_COMANDATE, NUM_POMPE_COMANDATE *)
  // as ST:
  //   _t1 := NOT TERZA_POMPA_COMANDATA AND NUM_POMPE_COMANDATE < NUM_POMPE_DA_COMANDARE AND P4_USABILE AND NOT P4_CMD;
  //   IF _t1 THEN P4_CMD := TRUE; END_IF;
  //   IF _t1 THEN NUM_POMPE_COMANDATE := NUM_POMPE_COMANDATE + 1; END_IF;
